(* PLC project MotorControl, AI-PLC-Integration AI SCL→LAD Generator 1.0 *)
(* stored: creationDateTime 2026-05-29T19:04:20.735391, modificationDateTime 2026-05-29T19:04:20.735391 *)

FUNCTION_BLOCK MotorControl
  VAR_INPUT
    bEmergencyStop : BOOL;  (* 急停（常闭触点） *)
    bStartForward : BOOL;  (* 正转启动按钮 *)
    bStop : BOOL;  (* 停止按钮（常闭） *)
    bStartReverse : BOOL;  (* 反转启动按钮 *)
    bOverload : BOOL;  (* 过载信号（常闭） *)
    bReset : BOOL;  (* 故障复位按钮 *)
  END_VAR
  VAR_OUTPUT
    bForwardOut : BOOL;  (* 正转输出 *)
    bReverseOut : BOOL;  (* 反转输出 *)
    bFault : BOOL;  (* 故障指示 *)
  END_VAR
  VAR
    bSafetyOK : BOOL;  (* 安全状态位（急停正常时=ON） *)
    bFaultLatch : BOOL;  (* 故障锁存位 *)
    bRunForward : BOOL;  (* 正转运行中间位 *)
    bRunReverse : BOOL;  (* 反转运行中间位 *)
  END_VAR
  VAR_TEMP
    tmrFeedback : TON;  (* 运行反馈超时定时器 *)
  END_VAR

(* LD diagram, written out as Structured Text *)
END_FUNCTION_BLOCK
